{attribute 'pack_mode' := '2'}
TYPE ST_XPU_STATE :
STRUCT
  Init            : E_XPU_INIT;
  State           : E_XPU_STATE;
  Check           : E_XPU_CHECK;  // cyclic check result
  DcLink          : BIT;          // power all motor modules is ON
END_STRUCT
END_TYPE

(* stored: Version 1.1.0.1
   DUT ST_XPU_STATE: Id {9176f11e-58d6-4e02-883d-244430cdaf5b} *)
